FUNCTION proj42_TupleStruct_3: BOOL
VAR_INPUT
    tuple: TupleStruct_3;
END_VAR


        proj42_TupleStruct_3 := tuple.field42;

END_FUNCTION

(* stored: ProductVersion 3.1.0.18, Version 1.1.0.1 *)
